// TIA Portal project "tank_doluluk_oranı" (V18)

(* hardware
DEVICE "S7-1200 station_1"  S7-1200 Station
   slot 0: "Rack_0"  S7-1200 Rack  Rack  V1.0
   slot 1: "PLC_1"  CPU 1214C AC/DC/Rly  6ES7 214-1BG40-0XB0  V4.6
*)

// ===== PLC "PLC_1"  CPU 1214C AC/DC/Rly =====

VAR_GLOBAL   // PLC tag table "Default tag table"
   "Tag_2" AT %Q0.1 : Bool;
   "Tag_3" AT %Q0.0 : Bool;
   "Tag_4" AT %Q0.2 : Bool;
   "ANALOG_GIRIS" AT %IW64 : Int;
END_VAR

ORGANIZATION_BLOCK "Main"   // OB1, LAD, ProgramCycle
TITLE = "Main Program Sweep (Cycle)"
{ S7_Optimized_Access := 'TRUE' }
VERSION : 0.1
// UYGULAMA 39: Bir tankin doluluk orani izlenecektir. Eger tank %80 ve üzerinde
// dolu ise Q 0.0, %20 ve altinda dolu ise Q 0.1 lambalari, doluluk orani bu iki deger
// arasinda ise Q0.2 lambasi yanacaktir. Tankin doluluk orani "O" ile "10" volt gerilim
// veren bir sensörden alinmaktadir.
// Tank %80 dolu ise 27648*0.80=22118 say: degerine tekabil eder.
// Tank %20 dolu ise 27648*0.20=5530 say: degerine tekabul eder.
   VAR_INPUT
      Initial_Call : Bool;   // Initial call of this OB
      Remanence : Bool;   // =True, if remanent data are available
   END_VAR
BEGIN

REGION Network 1
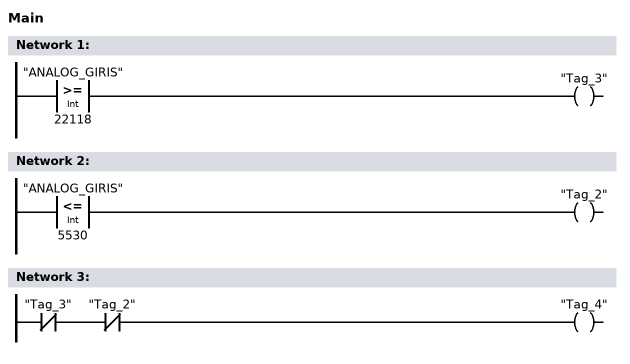
   RUNG wire#powerrail
      { S7_Templates := "SrcType := Int" } GE_Contact(in1 := "ANALOG_GIRIS", in2 := 22118)
      Coil( "Tag_3" )
   END_RUNG
   // the same network as SCL:
   "Tag_3" := "ANALOG_GIRIS" >= 22118;
END_REGION

REGION Network 2
   RUNG wire#powerrail
      { S7_Templates := "SrcType := Int" } LE_Contact(in1 := "ANALOG_GIRIS", in2 := 5530)
      Coil( "Tag_2" )
   END_RUNG
   // the same network as SCL:
   "Tag_2" := "ANALOG_GIRIS" <= 5530;
END_REGION

REGION Network 3
   RUNG wire#powerrail
      I_Contact( "Tag_3" )
      I_Contact( "Tag_2" )
      Coil( "Tag_4" )
   END_RUNG
   // the same network as SCL:
   "Tag_4" := NOT "Tag_3" AND NOT "Tag_2";
END_REGION
END_ORGANIZATION_BLOCK